TYPE ST_TopMoldProdPar_OLD :
STRUCT
	PositionDownSlow			: REAL;
	PositionDownCreep			: REAL; (*New sinds speed update*)
	PositionDownStop			: REAL;
END_STRUCT
END_TYPE

(* stored: Version 1.1.0.1, ProductVersion 3.1.4020.12
   DUT ST_TopMoldProdPar_OLD: Id {833b9db9-d468-444e-81eb-3e60e10f491c} *)
